Omron CX-Programmer project NewProject (CX-Programmer 9.73)

# PLC NewPLC1: CP1L M

## Global symbols (name address type ; comment)
0.00 BOOL  ; Start
0.03 BOOL  ; EMERGENCY
0.04 BOOL  ; Non metal Red
0.05 BOOL  ; Metal Blue
0.06 BOOL  ; Sensor
100.02 BOOL  ; BLUE BOX
100.03 BOOL  ; RED BOX
100.06 BOOL  ; Conveyor

## Program NewProgram1 (cyclic task 0)

### Section Section1

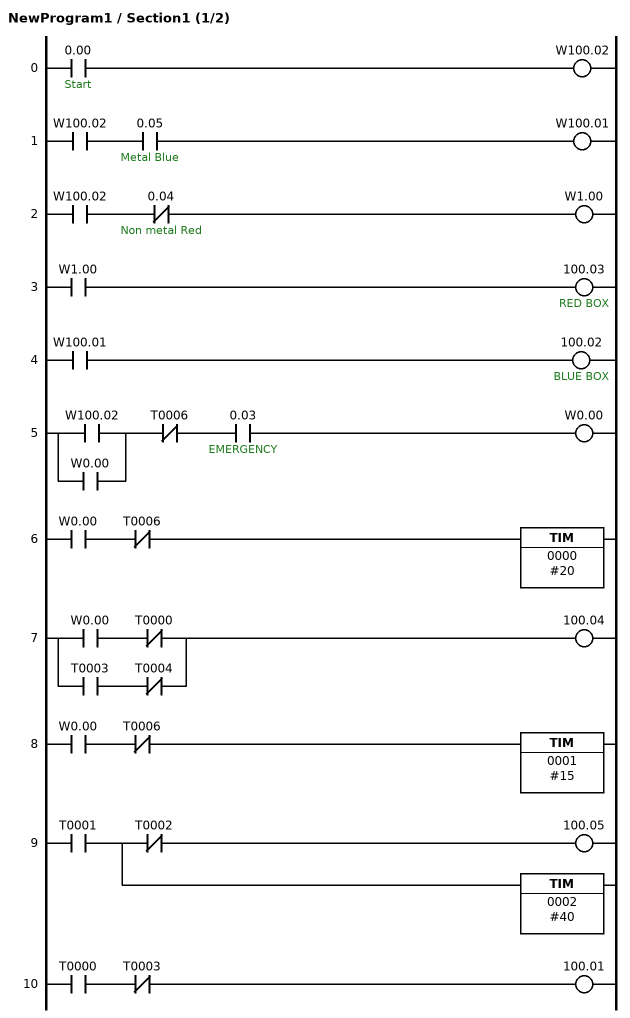
; rung 0
LD 0.00  ; Start
OUT W100.02
; rung 1
LD W100.02
AND 0.05  ; Metal Blue
OUT W100.01
; rung 2
LD W100.02
ANDNOT 0.04  ; Non metal Red
OUT W1.00
; rung 3
LD W1.00
OUT 100.03  ; RED BOX
; rung 4
LD W100.01
OUT 100.02  ; BLUE BOX
; rung 5
LD W100.02
OR W0.00
ANDNOT T0006
AND 0.03  ; EMERGENCY
OUT W0.00
; rung 6
LD W0.00
ANDNOT T0006
TIM 0000 #20
; rung 7
LD W0.00
ANDNOT T0000
LD T0003
ANDNOT T0004
ORLD
OUT 100.04
; rung 8
LD W0.00
ANDNOT T0006
TIM 0001 #15
; rung 9
LD T0001
OUT TR0
ANDNOT T0002
OUT 100.05
LD TR0
TIM 0002 #40
; rung 10
LD T0000
ANDNOT T0003
OUT 100.01

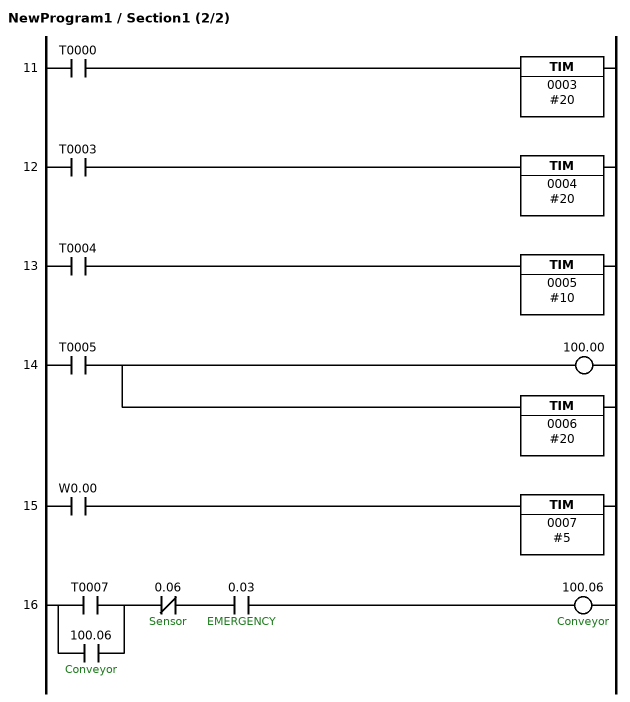
; rung 11
LD T0000
TIM 0003 #20
; rung 12
LD T0003
TIM 0004 #20
; rung 13
LD T0004
TIM 0005 #10
; rung 14
LD T0005
OUT 100.00
TIM 0006 #20
; rung 15
LD W0.00
TIM 0007 #5
; rung 16
LD T0007
OR 100.06  ; Conveyor
ANDNOT 0.06  ; Sensor
AND 0.03  ; EMERGENCY
OUT 100.06  ; Conveyor

### Section END
; rung 0
END(001)